(* PLC project RobotLibrarySysDep, Rexroth ctrlX PLC Engineering ctrlX PLC 2.6.6, author Thorsten Brach *)
(* stored: creationDateTime 2025-03-04T19:12:31.5427624, version 0.0.0.2, modificationDateTime 2025-03-04T19:09:29.8758205, organization Thorsten Brach *)
(* SRCI Robot Library System Dependencies *)

FUNCTION SysDepMemCmp : DINT
  VAR_INPUT
    pData1 : POINTER TO BYTE;  (* Pointer to 1st memory area to be compared with the 2nd memory area *)
    pData2 : POINTER TO BYTE;  (* Pointer to 2nd memory area to be compared with the 1st memory area *)
    DataLen : UDINT;  (* Amount of bytes to be compared *)
  END_VAR

            SysDepMemCmp := SysMemCmp( pBuffer1 := pData1, pBuffer2 := pData2, udiCount := DataLen );

          
END_FUNCTION

FUNCTION SysDepMemCpy : UDINT
  VAR_INPUT
    pDest : POINTER TO BYTE;  (* Pointer to memory address to be copied to (target) *)
    pSrc : POINTER TO BYTE;  (* Pointer to memory address to be copied from (source) *)
    DataLen : UDINT;  (* Amount of bytes to be copied *)
  END_VAR

            SysMemCpy( pDest := pDest, pSrc := pSrc, udiCount := DataLen );


          
END_FUNCTION

FUNCTION SysDepMemSet : UDINT
  VAR_INPUT
    pDest : POINTER TO BYTE;  (* Pointer to memory address to be filled (target) *)
    Value : BYTE;  (* Value with which the memory is to be initialized *)
    DataLen : UDINT;  (* Amount of bytes to be initialized in the memory block *)
  END_VAR

            SysMemSet( pDest := pDest, udiValue := Value, udiCount := DataLen );
          
END_FUNCTION

FUNCTION SysDepIsValidLReal : BOOL
  VAR_INPUT
    Value : LREAL;  (* Real value to validate *)
  END_VAR

            SysDepIsValidLReal := FPU.IsLRealNumber(Value);
          
END_FUNCTION

FUNCTION SysDepIsValidReal : BOOL
  VAR_INPUT
    Value : REAL;  (* Real value to validate *)
  END_VAR

            SysDepIsValidReal := FPU.IsRealNumber(Value);
          
END_FUNCTION
